SUBAPPLICATION T_FF_ILOCK_EVENT_AX (* Toggle-Flip-Flop mit Interlock / Reset-Eingang und SET-Event-Ausgang (AX Adapter Version) *)
  (* Standard: 61499-2; Description: Copyright (c) 2026 Meisterschulen am Ostbahnhof This program and the accompanying materials are made available under the terms of the Eclipse Public License 2.0 which is available at https://www.eclipse.org/legal/epl-2.0/ SPDX-License-Identifier: EPL-2.0 *)
  (* Version 1.0, 2026-09-10, Franz Höpfinger, Meisterschulen am Ostbahnhof, initial API and implementation (AX Adapter Version) *)
  PACKAGE MyLib::sys;
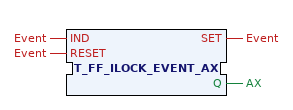
  EVENT_INPUT
    IND; (* Event Input (Clock / Click) *)
    RESET; (* External Reset Input *)
  END_EVENT
  EVENT_OUTPUT
    SET; (* Fired when switched ON (for Interlock reset of partner) *)
  END_EVENT
  PLUGS
    Q : adapter::types::unidirectional::AX; (* Adapter Output Q *)
  END_PLUGS
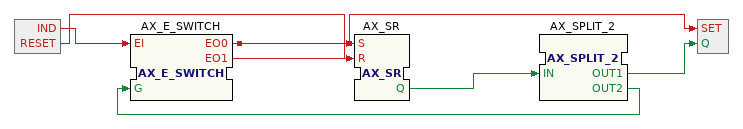
  FBS
    AX_E_SWITCH : adapter::events::unidirectional::AX_E_SWITCH;
    AX_SR : adapter::events::unidirectional::AX_SR;
    AX_SPLIT_2 : adapter::events::unidirectional::AX_SPLIT_2;
  END_FBS
  EVENT_CONNECTIONS
    IND TO AX_E_SWITCH.EI;
    AX_E_SWITCH.EO0 TO AX_SR.S;
    AX_E_SWITCH.EO0 TO SET;
    AX_E_SWITCH.EO1 TO AX_SR.R;
    RESET TO AX_SR.R;
  END_CONNECTIONS
  ADAPTER_CONNECTIONS
    AX_SR.Q TO AX_SPLIT_2.IN;
    AX_SPLIT_2.OUT1 TO Q;
    AX_SPLIT_2.OUT2 TO AX_E_SWITCH.G;
  END_CONNECTIONS
END_SUBAPPLICATION
